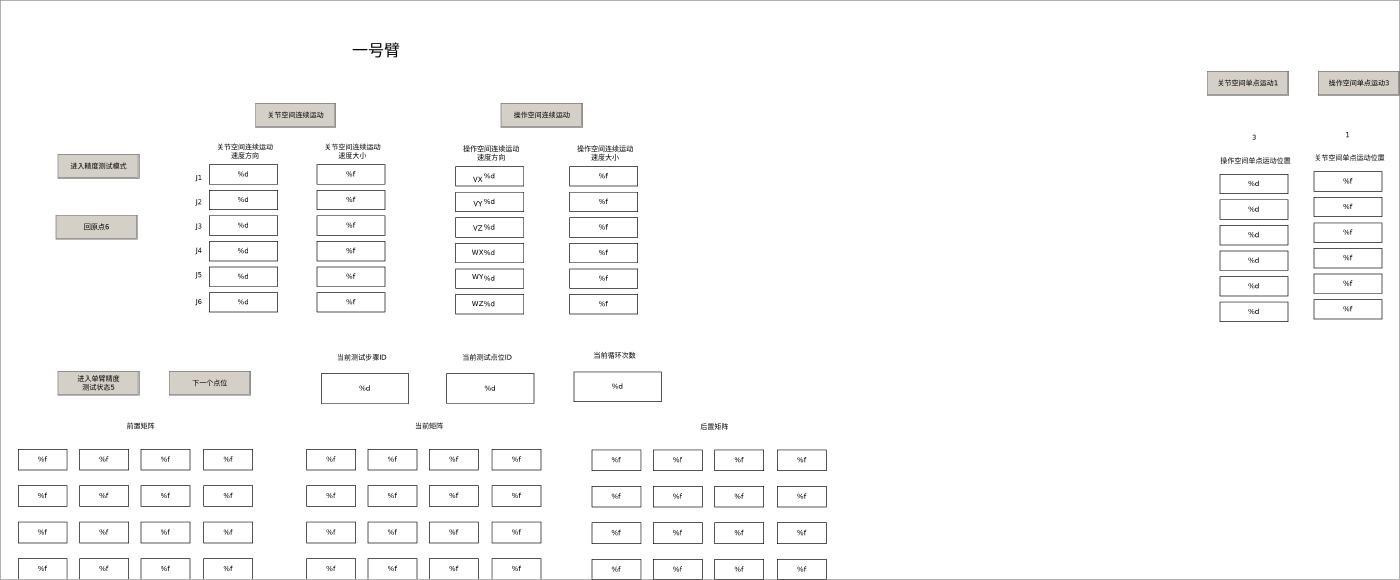
VISUALIZATION Robot_Jog_Arm1  // 2189x907
    Label (513,57 150x43), "一号臂"
    Rectangle (327,257 107x31), "%d", text variable: GVL_AccuracyTestVar.g_jntMotionDir[1][1]
        OnMouseClick: write the text variable via Default, min -1, max 1
    Label (308,222 150x29), "关节空间连续运动 速度方向"
    Rectangle (327,297 107x31), "%d", text variable: GVL_AccuracyTestVar.g_jntMotionDir[1][2]
        OnMouseClick: write the text variable via Default, min -1, max 1
    Rectangle (327,337 107x31), "%d", text variable: GVL_AccuracyTestVar.g_jntMotionDir[1][3]
        OnMouseClick: write the text variable via Default, min -1, max 1
    Rectangle (327,377 107x31), "%d", text variable: GVL_AccuracyTestVar.g_jntMotionDir[1][4]
        OnMouseClick: write the text variable via Default, min -1, max 1
    Rectangle (327,417 107x31), "%d", text variable: GVL_AccuracyTestVar.g_jntMotionDir[1][5]
        OnMouseClick: write the text variable via Default, min -1, max 1
    Rectangle (327,457 107x31), "%d", text variable: GVL_AccuracyTestVar.g_jntMotionDir[1][6]
        OnMouseClick: write the text variable via Default, min -1, max 1
    Group (2032,196 153x303), invisible if: TRUE
        Rectangle (22,72 107x31), "%f", text variable: GVL_AccuracyTestVar.g_targetJntPos[1][1]
            OnMouseClick: write the text variable via Default
        Label (3,36 150x30), "关节空间单点运动位置"
        Rectangle (22,112 107x31), "%f", text variable: GVL_AccuracyTestVar.g_targetJntPos[1][2]
            OnMouseClick: write the text variable via Default
        Rectangle (22,152 107x31), "%f", text variable: GVL_AccuracyTestVar.g_targetJntPos[1][3]
            OnMouseClick: write the text variable via Default
        Rectangle (22,192 107x31), "%f", text variable: GVL_AccuracyTestVar.g_targetJntPos[1][4]
            OnMouseClick: write the text variable via Default
        Rectangle (22,232 107x31), "%f", text variable: GVL_AccuracyTestVar.g_targetJntPos[1][5]
            OnMouseClick: write the text variable via Default
        Rectangle (22,272 107x31), "%f", text variable: GVL_AccuracyTestVar.g_targetJntPos[1][6]
            OnMouseClick: write the text variable via Default
        Label (0,0 150x30), "1"
    Rectangle (495,257 107x31), "%f", text variable: GVL_AccuracyTestVar.g_jntVel[1][1]
        OnMouseClick: write the text variable via Default
    Label (476,222 150x29), "关节空间连续运动 速度大小"
    Rectangle (495,297 107x31), "%f", text variable: GVL_AccuracyTestVar.g_jntVel[1][2]
        OnMouseClick: write the text variable via Default
    Rectangle (495,337 107x31), "%f", text variable: GVL_AccuracyTestVar.g_jntVel[1][3]
        OnMouseClick: write the text variable via Default
    Rectangle (495,377 107x31), "%f", text variable: GVL_AccuracyTestVar.g_jntVel[1][4]
        OnMouseClick: write the text variable via Default
    Rectangle (495,417 107x31), "%f", text variable: GVL_AccuracyTestVar.g_jntVel[1][5]
        OnMouseClick: write the text variable via Default
    Rectangle (495,457 107x31), "%f", text variable: GVL_AccuracyTestVar.g_jntVel[1][6]
        OnMouseClick: write the text variable via Default
    Group (1886,200 152x303), invisible if: TRUE
        Rectangle (21,72 107x31), "%d"
        Label (2,37 150x29), "操作空间单点运动位置"
        Rectangle (21,112 107x31), "%d"
        Rectangle (21,152 107x31), "%d"
        Rectangle (21,192 107x31), "%d"
        Rectangle (21,232 107x31), "%d"
        Rectangle (21,272 107x31), "%d"
        Label (0,0 150x30), "3"
    Rectangle (712,260 107x31), "%d", text variable: GVL_AccuracyTestVar.g_spatialMotionDir[1][1]
        OnMouseClick: write the text variable via Default, min -1, max 1
    Label (693,225 150x29), "操作空间连续运动 速度方向"
    Rectangle (712,300 107x31), "%d", text variable: GVL_AccuracyTestVar.g_spatialMotionDir[1][2]
        OnMouseClick: write the text variable via Default, min -1, max 1
    Rectangle (712,340 107x31), "%d", text variable: GVL_AccuracyTestVar.g_spatialMotionDir[1][3]
        OnMouseClick: write the text variable via Default, min -1, max 1
    Rectangle (712,380 107x31), "%d", text variable: GVL_AccuracyTestVar.g_spatialMotionDir[1][4]
        OnMouseClick: write the text variable via Default, min -1, max 1
    Rectangle (712,420 107x31), "%d", text variable: GVL_AccuracyTestVar.g_spatialMotionDir[1][5]
        OnMouseClick: write the text variable via Default, min -1, max 1
    Rectangle (712,460 107x31), "%d", text variable: GVL_AccuracyTestVar.g_spatialMotionDir[1][6]
        OnMouseClick: write the text variable via Default, min -1, max 1
    Rectangle (890,260 107x31), "%f", text variable: GVL_AccuracyTestVar.g_spatialVel[1][1]
        OnMouseClick: write the text variable via Default
    Label (871,225 150x29), "操作空间连续运动 速度大小"
    Rectangle (890,300 107x31), "%f", text variable: GVL_AccuracyTestVar.g_spatialVel[1][2]
        OnMouseClick: write the text variable via Default
    Rectangle (890,340 107x31), "%f", text variable: GVL_AccuracyTestVar.g_spatialVel[1][3]
        OnMouseClick: write the text variable via Default
    Rectangle (890,380 107x31), "%f", text variable: GVL_AccuracyTestVar.g_spatialVel[1][4]
        OnMouseClick: write the text variable via Default
    Rectangle (890,420 107x31), "%f", text variable: GVL_AccuracyTestVar.g_spatialVel[1][5]
        OnMouseClick: write the text variable via Default
    Rectangle (890,460 107x31), "%f", text variable: GVL_AccuracyTestVar.g_spatialVel[1][6]
        OnMouseClick: write the text variable via Default
    Button (90,241 128x38), "进入精度测试模式", colour toggle: GVL_AccuracyTestVar.g_enterPrecisionTestMode[1]
        toggle GVL_AccuracyTestVar.g_enterPrecisionTestMode[1]
    Group (1887,111 302x38), invisible if: TRUE
        Button (0,0 128x38), "关节空间单点运动1", colour toggle: A1_Arm1ModeL[1,1]
            tap A1_Arm1Mode[1,1]
        Button (174,0 128x38), "操作空间单点运动3", colour toggle: A1_Arm1ModeL[1,3]
            tap A1_Arm1Mode[1,3]
    Button (399,161 126x38), "关节空间连续运动", colour toggle: A1_Arm1ModeL[1,2]
        tap A1_Arm1Mode[1,2]
    Button (783,161 128x38), "操作空间连续运动", colour toggle: A1_Arm1ModeL[1,4]
        tap A1_Arm1Mode[1,4]
    Button (87,336 128x38), "回原点6", colour toggle: A1_Arm1ModeL[1,6]
        tap A1_Arm1Mode[1,6]
    Button (90,580 128x38), "进入单臂精度 测试状态5", colour toggle: A1_Arm1ModeL[1,5]
        tap A1_Arm1Mode[1,5]
    Button (264,580 128x38), "下一个点位", colour toggle: GVL_AccuracyTestVar.g_nextStep[1]
        tap GVL_AccuracyTestVar.g_nextStep[1]
    Rectangle (502,584 137x47), "%d", text variable: GVL_AccuracyTestVar.g_curStep[1]
    Label (491,544 150x30), "当前测试步骤ID"
    Rectangle (698,584 137x47), "%d", text variable: GVL_AccuracyTestVar.g_testPointId[1]
    Label (687,544 150x30), "当前测试点位ID"
    Rectangle (897,581 137x47), "%d", text variable: GVL_AccuracyTestVar.g_testCycleId[1]
    Label (886,541 150x30), "当前循环次数"
    Group (304,263 14x224)
        Label (0,0 14x30), "J1"
        Label (0,38 14x30), "J2"
        Label (0,76 14x30), "J3"
        Label (0,114 14x30), "J4"
        Label (0,152 14x30), "J5"
        Label (0,194 14x30), "J6"
    Group (672,266 26x224)
        Label (0,0 150x30), "VX"
        Label (0,38 150x30), "VY"
        Label (0,76 150x30), "VZ"
        Label (0,114 150x30), "WX"
        Label (0,152 150x30), "WY"
        Label (0,194 150x30), "WZ"
    Label (145,652 150x29), "前置矩阵"
    Rectangle (28,702 77x33), "%f", text variable: GVL_AccuracyTestVar.g_frontPose[1].m_rot[1,1]
    Rectangle (124,702 77x33), "%f", text variable: GVL_AccuracyTestVar.g_frontPose[1].m_rot[1,2]
    Rectangle (220,702 77x33), "%f", text variable: GVL_AccuracyTestVar.g_frontPose[1].m_rot[1,3]
    Rectangle (318,702 77x33), "%f", text variable: GVL_AccuracyTestVar.g_frontPose[1].m_pos[1]
    Rectangle (28,759 77x33), "%f", text variable: GVL_AccuracyTestVar.g_frontPose[1].m_rot[2,1]
    Rectangle (28,816 77x33), "%f", text variable: GVL_AccuracyTestVar.g_frontPose[1].m_rot[3,1]
    Rectangle (28,873 77x33), "%f", text variable: 0
    Rectangle (124,759 77x33), "%f", text variable: GVL_AccuracyTestVar.g_frontPose[1].m_rot[2,2]
    Rectangle (220,759 77x33), "%f", text variable: GVL_AccuracyTestVar.g_frontPose[1].m_rot[2,3]
    Rectangle (318,759 77x33), "%f", text variable: GVL_AccuracyTestVar.g_frontPose[1].m_pos[2]
    Rectangle (124,816 77x33), "%f", text variable: GVL_AccuracyTestVar.g_frontPose[1].m_rot[3,2]
    Rectangle (220,816 77x33), "%f", text variable: GVL_AccuracyTestVar.g_frontPose[1].m_rot[3,3]
    Rectangle (318,816 77x33), "%f", text variable: GVL_AccuracyTestVar.g_frontPose[1].m_pos[3]
    Rectangle (124,873 77x33), "%f", text variable: 0
    Rectangle (220,873 77x33), "%f", text variable: 0
    Rectangle (318,873 77x33), "%f", text variable: 1
    Label (596,652 150x29), "当前矩阵"
    Rectangle (479,702 77x33), "%f", text variable: GVL_AccuracyTestVar.g_slaveArmPose[1].m_rot[1,1]
    Rectangle (575,702 77x33), "%f", text variable: GVL_AccuracyTestVar.g_slaveArmPose[1].m_rot[1,2]
    Rectangle (671,702 77x33), "%f", text variable: GVL_AccuracyTestVar.g_slaveArmPose[1].m_rot[1,3]
    Rectangle (769,702 77x33), "%f", text variable: GVL_AccuracyTestVar.g_slaveArmPose[1].m_pos[1]
    Rectangle (479,759 77x33), "%f", text variable: GVL_AccuracyTestVar.g_slaveArmPose[1].m_rot[2,1]
    Rectangle (479,816 77x33), "%f", text variable: GVL_AccuracyTestVar.g_slaveArmPose[1].m_rot[3,1]
    Rectangle (479,873 77x33), "%f", text variable: 0
    Rectangle (575,759 77x33), "%f", text variable: GVL_AccuracyTestVar.g_slaveArmPose[1].m_rot[2,2]
    Rectangle (671,759 77x33), "%f", text variable: GVL_AccuracyTestVar.g_slaveArmPose[1].m_rot[2,3]
    Rectangle (769,759 77x33), "%f", text variable: GVL_AccuracyTestVar.g_slaveArmPose[1].m_pos[2]
    Rectangle (575,816 77x33), "%f", text variable: GVL_AccuracyTestVar.g_slaveArmPose[1].m_rot[3,2]
    Rectangle (671,816 77x33), "%f", text variable: GVL_AccuracyTestVar.g_slaveArmPose[1].m_rot[3,3]
    Rectangle (769,816 77x33), "%f", text variable: GVL_AccuracyTestVar.g_slaveArmPose[1].m_pos[3]
    Rectangle (575,873 77x33), "%f", text variable: 0
    Rectangle (671,873 77x33), "%f", text variable: 0
    Rectangle (769,873 77x33), "%f", text variable: 1
    Label (1042,653 150x29), "后置矩阵"
    Rectangle (925,703 77x33), "%f", text variable: GVL_AccuracyTestVar.g_endPose[1].m_rot[1,1]
    Rectangle (1021,703 77x33), "%f", text variable: GVL_AccuracyTestVar.g_endPose[1].m_rot[1,2]
    Rectangle (1117,703 77x33), "%f", text variable: GVL_AccuracyTestVar.g_endPose[1].m_rot[1,3]
    Rectangle (1215,703 77x33), "%f", text variable: GVL_AccuracyTestVar.g_endPose[1].m_pos[1]
    Rectangle (925,760 77x33), "%f", text variable: GVL_AccuracyTestVar.g_endPose[1].m_rot[2,1]
    Rectangle (925,817 77x33), "%f", text variable: GVL_AccuracyTestVar.g_endPose[1].m_rot[3,1]
    Rectangle (925,874 77x33), "%f", text variable: 0
    Rectangle (1021,760 77x33), "%f", text variable: GVL_AccuracyTestVar.g_endPose[1].m_rot[2,2]
    Rectangle (1117,760 77x33), "%f", text variable: GVL_AccuracyTestVar.g_endPose[1].m_rot[2,3]
    Rectangle (1215,760 77x33), "%f", text variable: GVL_AccuracyTestVar.g_endPose[1].m_pos[2]
    Rectangle (1021,817 77x33), "%f", text variable: GVL_AccuracyTestVar.g_endPose[1].m_rot[3,2]
    Rectangle (1117,817 77x33), "%f", text variable: GVL_AccuracyTestVar.g_endPose[1].m_rot[3,3]
    Rectangle (1215,817 77x33), "%f", text variable: GVL_AccuracyTestVar.g_frontPose[1].m_pos[3]
    Rectangle (1021,874 77x33), "%f", text variable: 0
    Rectangle (1117,874 77x33), "%f", text variable: 0
    Rectangle (1215,874 77x33), "%f", text variable: 1
END_VISUALIZATION

(* stored: Version 1.1.0.1, ProductVersion 3.1.4024.11
   Visu Robot_Jog_Arm1: Id {c275d056-9c8b-436c-b15b-86e3d9a625b0} *)
